# EPICS autosave request: services/bl11t-ea-multi-01/config/ETLdetector_settings.req
$(P)$(Q):UPDATE.SCAN
